                                        FB_Bacnet.StartStopCommand_145.bEnWrite := TRUE;
                                        FB_Bacnet.StartStopCommand_145.bVal := TRUE;
                                    19: 
                                        
                                        FB_Bacnet.StartStopCommand_146.bEnWrite := TRUE;
                                        FB_Bacnet.StartStopCommand_146.bVal := TRUE;
                                    20: 
                                        
                                        FB_Bacnet.StartStopCommand_147.bEnWrite := TRUE;
                                        FB_Bacnet.StartStopCommand_147.bVal := TRUE;
                                    21: 
                                        
                                        FB_Bacnet.StartStopCommand_148.bEnWrite := TRUE;
                                        FB_Bacnet.StartStopCommand_148.bVal := TRUE;
                                    22: 
                                        
                                        FB_Bacnet.StartStopCommand_176.bEnWrite := TRUE;
                                        FB_Bacnet.StartStopCommand_176.bVal := TRUE;
                                    23: 
                                        //FB_Bacnet.StartStopCommand_177.bEnWrite := TRUE;
                                        //FB_Bacnet.StartStopCommand_177.bVal := TRUE;
                                END_CASE
                            END_IF
                        END_FOR
                    END_IF
                    // Schedule Unit OFF
                    IF wSchedWEHourEndF2_ = currH AND wSchedWEMinEndF2_ = currM AND NOT bUnitTriggered THEN
                        bUnitTriggered := TRUE;
                        FOR i := 1 TO 23 DO
                            // Send command unit OFF
                            IF bUnitF2_[i] THEN 
                                CASE i OF
                                    1: 
                                        
                                        FB_Bacnet.StartStopCommand_128.bEnWrite := TRUE;
                                        FB_Bacnet.StartStopCommand_128.bVal := FALSE;
                                    2: 
                                        
                                        FB_Bacnet.StartStopCommand_129.bEnWrite := TRUE;
                                        FB_Bacnet.StartStopCommand_129.bVal := FALSE;
                                    3: 
                                        
                                        FB_Bacnet.StartStopCommand_130.bEnWrite := TRUE;
                                        FB_Bacnet.StartStopCommand_130.bVal := FALSE;
                                    4: 
                                        
                                        FB_Bacnet.StartStopCommand_131.bEnWrite := TRUE;
                                        FB_Bacnet.StartStopCommand_131.bVal := FALSE;
                                    5: 
                                        
                                        FB_Bacnet.StartStopCommand_132.bEnWrite := TRUE;
                                        FB_Bacnet.StartStopCommand_132.bVal := FALSE;
                                    6: 
                                        
                                        FB_Bacnet.StartStopCommand_133.bEnWrite := TRUE;
                                        FB_Bacnet.StartStopCommand_133.bVal := FALSE;
                                    7: 
                                        
                                        FB_Bacnet.StartStopCommand_134.bEnWrite := TRUE;
                                        FB_Bacnet.StartStopCommand_134.bVal := FALSE;
                                    8: 
                                        
                                        FB_Bacnet.StartStopCommand_135.bEnWrite := TRUE;
                                        FB_Bacnet.StartStopCommand_135.bVal := FALSE;
                                    9: 
                                        
                                        FB_Bacnet.StartStopCommand_136.bEnWrite := TRUE;
                                        FB_Bacnet.StartStopCommand_136.bVal := FALSE;
                                    10: 
                                        
                                        FB_Bacnet.StartStopCommand_137.bEnWrite := TRUE;
                                        FB_Bacnet.StartStopCommand_137.bVal := FALSE;
                                    11: 
                                        
                                        FB_Bacnet.StartStopCommand_138.bEnWrite := TRUE;
                                        FB_Bacnet.StartStopCommand_138.bVal := FALSE;
                                    12: 
                                        
                                        FB_Bacnet.StartStopCommand_139.bEnWrite := TRUE;
                                        FB_Bacnet.StartStopCommand_139.bVal := FALSE;
                                    13: 
                                        //FB_Bacnet.StartStopCommand_140.bEnWrite := TRUE;
                                        //FB_Bacnet.StartStopCommand_140.bVal := FALSE;
                                    14: 
                                        
                                        FB_Bacnet.StartStopCommand_141.bEnWrite := TRUE;
                                        FB_Bacnet.StartStopCommand_141.bVal := FALSE;
                                    15: 
                                        
                                        FB_Bacnet.StartStopCommand_142.bEnWrite := TRUE;
                                        FB_Bacnet.StartStopCommand_142.bVal := FALSE;
                                    16: 
                                        
                                        FB_Bacnet.StartStopCommand_143.bEnWrite := TRUE;
                                        FB_Bacnet.StartStopCommand_143.bVal := FALSE;
                                    17: 
                                        
                                        FB_Bacnet.StartStopCommand_144.bEnWrite := TRUE;
                                        FB_Bacnet.StartStopCommand_144.bVal := FALSE;
                                    18: 
                                        
                                        FB_Bacnet.StartStopCommand_145.bEnWrite := TRUE;
                                        FB_Bacnet.StartStopCommand_145.bVal := FALSE;
                                    19: 
                                        
                                        FB_Bacnet.StartStopCommand_146.bEnWrite := TRUE;
                                        FB_Bacnet.StartStopCommand_146.bVal := FALSE;
                                    20: 
                                        
                                        FB_Bacnet.StartStopCommand_147.bEnWrite := TRUE;
                                        FB_Bacnet.StartStopCommand_147.bVal := FALSE;
                                    21: 
                                        
                                        FB_Bacnet.StartStopCommand_148.bEnWrite := TRUE;
                                        FB_Bacnet.StartStopCommand_148.bVal := FALSE;
                                    22: 
                                        
                                        FB_Bacnet.StartStopCommand_176.bEnWrite := TRUE;
                                        FB_Bacnet.StartStopCommand_176.bVal := FALSE;
                                    23: 
                                        //FB_Bacnet.StartStopCommand_177.bEnWrite := TRUE;
                                        //FB_Bacnet.StartStopCommand_177.bVal := FALSE;
                                END_CASE
                            END_IF
                        END_FOR
                    END_IF
                END_IF
            END_IF
        END_IF

END_FUNCTION_BLOCK

// ---- POUs/FB_Scheduler/FB_Scheduler_F3.TcPOU

      FUNCTION_BLOCK FB_Scheduler_F3
      VAR_INPUT
          currH : WORD;
          currM : WORD;
          currD : WORD;
      END_VAR
      VAR_IN_OUT
          FB_Bacnet : FB_BACnet_DAIKIN_MasterStation_III_No_1;
      END_VAR
      VAR
          i : INT;
          bUnitTriggered : BOOL := FALSE; // New flag to track execution
          prevMinute : WORD := 0;        // New variable to track the previous minute
      END_VAR
      VAR PERSISTENT
          //scheduler var
          bEnSchedF3_ : BOOL := FALSE;
          wSchedWDHourStartF3_ : WORD; 
          wSchedWDMinStartF3_ : WORD; 
          wSchedWEHourStartF3_ : WORD; 
          wSchedWEMinStartF3_ : WORD;
          wSchedWDHourEndF3_ : WORD;
          wSchedWDMinEndF3_ : WORD;
          wSchedWEHourEndF3_ : WORD;
          wSchedWEMinEndF3_ : WORD;
          //unit var
          bUnitF3_ : ARRAY [1..22] OF BOOL;
      END_VAR


        // Reset trigger flag at minute change or at the exact scheduled time
        IF currM <> prevMinute OR 
           (currH = wSchedWDHourStartF3_ AND currM = wSchedWDMinStartF3_) OR 
           (currH = wSchedWDHourEndF3_ AND currM = wSchedWDMinEndF3_) THEN
            bUnitTriggered := FALSE;
            prevMinute := currM;
        END_IF

        // Unit Schedule Enable
        IF bEnSchedF3_ THEN
            // Weekday schedule
            IF currD >= 1 AND currD <= 5 THEN
                IF (wSchedWDHourStartF3_ <> wSchedWDHourEndF3_ OR wSchedWDMinStartF3_ <> wSchedWDMinEndF3_) THEN
                    // Schedule Unit ON
                    IF wSchedWDHourStartF3_ = currH AND wSchedWDMinStartF3_ = currM AND NOT bUnitTriggered THEN
                        bUnitTriggered := TRUE;
                        FOR i := 1 TO 22 DO
                            // Send command unit ON
                            IF bUnitF3_[i] THEN 
                                CASE i OF
                                    1: 

                                        //FB_Bacnet.StartStopCommand_192.bEnWrite := TRUE;
                                        //FB_Bacnet.StartStopCommand_192.bVal := TRUE;
                                    2: 
                                        
                                        FB_Bacnet.StartStopCommand_193.bEnWrite := TRUE;
                                        FB_Bacnet.StartStopCommand_193.bVal := TRUE;
                                    3: 
                                        
                                        FB_Bacnet.StartStopCommand_194.bEnWrite := TRUE;
                                        FB_Bacnet.StartStopCommand_194.bVal := TRUE;
                                    4: 
                                        
                                        FB_Bacnet.StartStopCommand_195.bEnWrite := TRUE;
                                        FB_Bacnet.StartStopCommand_195.bVal := TRUE;
                                    5: 
                                        
                                        FB_Bacnet.StartStopCommand_196.bEnWrite := TRUE;
                                        FB_Bacnet.StartStopCommand_196.bVal := TRUE;
                                    6: 
                                        
                                        FB_Bacnet.StartStopCommand_197.bEnWrite := TRUE;
                                        FB_Bacnet.StartStopCommand_197.bVal := TRUE;
                                    7: 
                                        
                                        FB_Bacnet.StartStopCommand_198.bEnWrite := TRUE;
                                        FB_Bacnet.StartStopCommand_198.bVal := TRUE;
                                    8: 
                                        
                                        FB_Bacnet.StartStopCommand_199.bEnWrite := TRUE;
                                        FB_Bacnet.StartStopCommand_199.bVal := TRUE;
                                    9: 
                                        
                                        FB_Bacnet.StartStopCommand_200.bEnWrite := TRUE;
                                        FB_Bacnet.StartStopCommand_200.bVal := TRUE;
                                    10: 
                                        
                                        FB_Bacnet.StartStopCommand_201.bEnWrite := TRUE;
                                        FB_Bacnet.StartStopCommand_201.bVal := TRUE;
                                    11: 
                                        
                                        FB_Bacnet.StartStopCommand_202.bEnWrite := TRUE;
                                        FB_Bacnet.StartStopCommand_202.bVal := TRUE;
                                    12: 
                                        
                                        FB_Bacnet.StartStopCommand_203.bEnWrite := TRUE;
                                        FB_Bacnet.StartStopCommand_203.bVal := TRUE;
                                    13: 
                                        
                                        FB_Bacnet.StartStopCommand_204.bEnWrite := TRUE;
                                        FB_Bacnet.StartStopCommand_204.bVal := TRUE;
                                    14: 
                                        
                                        FB_Bacnet.StartStopCommand_205.bEnWrite := TRUE;
                                        FB_Bacnet.StartStopCommand_205.bVal := TRUE;
                                    15: 
                                        
                                        FB_Bacnet.StartStopCommand_206.bEnWrite := TRUE;
                                        FB_Bacnet.StartStopCommand_206.bVal := TRUE;
                                    16: 
                                        
                                        FB_Bacnet.StartStopCommand_207.bEnWrite := TRUE;
                                        FB_Bacnet.StartStopCommand_207.bVal := TRUE;
                                    17: 
                                        
                                        FB_Bacnet.StartStopCommand_208.bEnWrite := TRUE;
                                        FB_Bacnet.StartStopCommand_208.bVal := TRUE;
                                    18: 
                                        
                                        FB_Bacnet.StartStopCommand_209.bEnWrite := TRUE;
                                        FB_Bacnet.StartStopCommand_209.bVal := TRUE;
                                    19: 
                                        
                                        FB_Bacnet.StartStopCommand_210.bEnWrite := TRUE;
                                        FB_Bacnet.StartStopCommand_210.bVal := TRUE;
                                    20: 
                                        
                                        FB_Bacnet.StartStopCommand_211.bEnWrite := TRUE;
                                        FB_Bacnet.StartStopCommand_211.bVal := TRUE;
                                    21: 
                                        
                                        FB_Bacnet.StartStopCommand_212.bEnWrite := TRUE;
                                        FB_Bacnet.StartStopCommand_212.bVal := TRUE;
                                    22: 
                                        
                                        FB_Bacnet.StartStopCommand_224.bEnWrite := TRUE;
                                        FB_Bacnet.StartStopCommand_224.bVal := TRUE;
                                END_CASE
                            END_IF
                        END_FOR
                    END_IF
                    // Schedule Unit OFF
                    IF wSchedWDHourEndF3_ = currH AND wSchedWDMinEndF3_ = currM AND NOT bUnitTriggered THEN
                        bUnitTriggered := TRUE;
                        FOR i := 1 TO 22 DO
                            // Send command unit OFF
                            IF bUnitF3_[i] THEN 
                                CASE i OF
                                    1: 

                                        //FB_Bacnet.StartStopCommand_192.bEnWrite := TRUE;
                                        //FB_Bacnet.StartStopCommand_192.bVal := FALSE;
                                    2: 
                                        
                                        FB_Bacnet.StartStopCommand_193.bEnWrite := TRUE;
                                        FB_Bacnet.StartStopCommand_193.bVal := FALSE;
                                    3: 
                                        
                                        FB_Bacnet.StartStopCommand_194.bEnWrite := TRUE;
                                        FB_Bacnet.StartStopCommand_194.bVal := FALSE;
                                    4: 
                                        
                                        FB_Bacnet.StartStopCommand_195.bEnWrite := TRUE;
                                        FB_Bacnet.StartStopCommand_195.bVal := FALSE;
                                    5: 
                                        
                                        FB_Bacnet.StartStopCommand_196.bEnWrite := TRUE;
                                        FB_Bacnet.StartStopCommand_196.bVal := FALSE;
                                    6: 
                                        
                                        FB_Bacnet.StartStopCommand_197.bEnWrite := TRUE;
                                        FB_Bacnet.StartStopCommand_197.bVal := FALSE;
                                    7: 
                                        
                                        FB_Bacnet.StartStopCommand_198.bEnWrite := TRUE;
                                        FB_Bacnet.StartStopCommand_198.bVal := FALSE;
                                    8: 
                                        
                                        FB_Bacnet.StartStopCommand_199.bEnWrite := TRUE;
                                        FB_Bacnet.StartStopCommand_199.bVal := FALSE;
                                    9: 
                                        
                                        FB_Bacnet.StartStopCommand_200.bEnWrite := TRUE;
                                        FB_Bacnet.StartStopCommand_200.bVal := FALSE;
                                    10: 
                                        
                                        FB_Bacnet.StartStopCommand_201.bEnWrite := TRUE;
                                        FB_Bacnet.StartStopCommand_201.bVal := FALSE;
                                    11: 
                                        
                                        FB_Bacnet.StartStopCommand_202.bEnWrite := TRUE;
                                        FB_Bacnet.StartStopCommand_202.bVal := FALSE;
                                    12: 
                                        
                                        FB_Bacnet.StartStopCommand_203.bEnWrite := TRUE;
                                        FB_Bacnet.StartStopCommand_203.bVal := FALSE;
                                    13: 
                                        
                                        FB_Bacnet.StartStopCommand_204.bEnWrite := TRUE;
                                        FB_Bacnet.StartStopCommand_204.bVal := FALSE;
                                    14: 
                                        
                                        FB_Bacnet.StartStopCommand_205.bEnWrite := TRUE;
                                        FB_Bacnet.StartStopCommand_205.bVal := FALSE;
                                    15: 
                                        
                                        FB_Bacnet.StartStopCommand_206.bEnWrite := TRUE;
                                        FB_Bacnet.StartStopCommand_206.bVal := FALSE;
                                    16: 
                                        
                                        FB_Bacnet.StartStopCommand_207.bEnWrite := TRUE;
                                        FB_Bacnet.StartStopCommand_207.bVal := FALSE;
                                    17: 
                                        
                                        FB_Bacnet.StartStopCommand_208.bEnWrite := TRUE;
                                        FB_Bacnet.StartStopCommand_208.bVal := FALSE;
                                    18: 
                                        
                                        FB_Bacnet.StartStopCommand_209.bEnWrite := TRUE;
                                        FB_Bacnet.StartStopCommand_209.bVal := FALSE;
                                    19: 
                                        
                                        FB_Bacnet.StartStopCommand_210.bEnWrite := TRUE;
                                        FB_Bacnet.StartStopCommand_210.bVal := FALSE;
                                    20: 
                                        
                                        FB_Bacnet.StartStopCommand_211.bEnWrite := TRUE;
                                        FB_Bacnet.StartStopCommand_211.bVal := FALSE;
                                    21: 
                                        
                                        FB_Bacnet.StartStopCommand_212.bEnWrite := TRUE;
                                        FB_Bacnet.StartStopCommand_212.bVal := FALSE;
                                    22: 
                                        
                                        FB_Bacnet.StartStopCommand_224.bEnWrite := TRUE;
                                        FB_Bacnet.StartStopCommand_224.bVal := FALSE;
                                END_CASE
                            END_IF
                        END_FOR
                    END_IF
                END_IF
            END_IF

            // Weekend schedule
            IF currD = 0 OR currD = 6 THEN
                IF (wSchedWEHourStartF3_ <> wSchedWEHourEndF3_ OR wSchedWEMinStartF3_ <> wSchedWEMinEndF3_) THEN
                    // Schedule Unit ON
                    IF wSchedWEHourStartF3_ = currH AND wSchedWEMinStartF3_ = currM AND NOT bUnitTriggered THEN
                        bUnitTriggered := TRUE;
                        FOR i := 1 TO 22 DO
                            // Send command unit ON
                            IF bUnitF3_[i] THEN 
                                CASE i OF
                                    1: 

                                        //FB_Bacnet.StartStopCommand_192.bEnWrite := TRUE;
                                        //FB_Bacnet.StartStopCommand_192.bVal := TRUE;
                                    2: 
                                        
                                        FB_Bacnet.StartStopCommand_193.bEnWrite := TRUE;
                                        FB_Bacnet.StartStopCommand_193.bVal := TRUE;
                                    3: 
                                        
                                        FB_Bacnet.StartStopCommand_194.bEnWrite := TRUE;
                                        FB_Bacnet.StartStopCommand_194.bVal := TRUE;
                                    4: 
                                        
                                        FB_Bacnet.StartStopCommand_195.bEnWrite := TRUE;
                                        FB_Bacnet.StartStopCommand_195.bVal := TRUE;
                                    5: 
                                        
                                        FB_Bacnet.StartStopCommand_196.bEnWrite := TRUE;
                                        FB_Bacnet.StartStopCommand_196.bVal := TRUE;
                                    6: 
                                        
                                        FB_Bacnet.StartStopCommand_197.bEnWrite := TRUE;
                                        FB_Bacnet.StartStopCommand_197.bVal := TRUE;
                                    7: 
                                        
                                        FB_Bacnet.StartStopCommand_198.bEnWrite := TRUE;
                                        FB_Bacnet.StartStopCommand_198.bVal := TRUE;
                                    8: 
                                        
                                        FB_Bacnet.StartStopCommand_199.bEnWrite := TRUE;
                                        FB_Bacnet.StartStopCommand_199.bVal := TRUE;
                                    9: 
                                        
                                        FB_Bacnet.StartStopCommand_200.bEnWrite := TRUE;
                                        FB_Bacnet.StartStopCommand_200.bVal := TRUE;
                                    10: 
                                        
                                        FB_Bacnet.StartStopCommand_201.bEnWrite := TRUE;
                                        FB_Bacnet.StartStopCommand_201.bVal := TRUE;
                                    11: 
                                        
                                        FB_Bacnet.StartStopCommand_202.bEnWrite := TRUE;
                                        FB_Bacnet.StartStopCommand_202.bVal := TRUE;
                                    12: 
                                        
                                        FB_Bacnet.StartStopCommand_203.bEnWrite := TRUE;
                                        FB_Bacnet.StartStopCommand_203.bVal := TRUE;
                                    13: 
                                        
                                        FB_Bacnet.StartStopCommand_204.bEnWrite := TRUE;
                                        FB_Bacnet.StartStopCommand_204.bVal := TRUE;
                                    14: 
                                        
                                        FB_Bacnet.StartStopCommand_205.bEnWrite := TRUE;
                                        FB_Bacnet.StartStopCommand_205.bVal := TRUE;
                                    15: 
                                        
                                        FB_Bacnet.StartStopCommand_206.bEnWrite := TRUE;
                                        FB_Bacnet.StartStopCommand_206.bVal := TRUE;
                                    16: 
                                        
                                        FB_Bacnet.StartStopCommand_207.bEnWrite := TRUE;
                                        FB_Bacnet.StartStopCommand_207.bVal := TRUE;
                                    17: 
                                        
                                        FB_Bacnet.StartStopCommand_208.bEnWrite := TRUE;
                                        FB_Bacnet.StartStopCommand_208.bVal := TRUE;
                                    18: 
                                        
                                        FB_Bacnet.StartStopCommand_209.bEnWrite := TRUE;
                                        FB_Bacnet.StartStopCommand_209.bVal := TRUE;
                                    19: 
                                        
                                        FB_Bacnet.StartStopCommand_210.bEnWrite := TRUE;
                                        FB_Bacnet.StartStopCommand_210.bVal := TRUE;
                                    20: 
                                        
                                        FB_Bacnet.StartStopCommand_211.bEnWrite := TRUE;
                                        FB_Bacnet.StartStopCommand_211.bVal := TRUE;
                                    21: 
                                        
                                        FB_Bacnet.StartStopCommand_212.bEnWrite := TRUE;
                                        FB_Bacnet.StartStopCommand_212.bVal := TRUE;
                                    22: 
                                        
                                        FB_Bacnet.StartStopCommand_224.bEnWrite := TRUE;
                                        FB_Bacnet.StartStopCommand_224.bVal := TRUE;
                                END_CASE
                            END_IF
                        END_FOR
                    END_IF
                    // Schedule Unit OFF
                    IF wSchedWEHourEndF3_ = currH AND wSchedWEMinEndF3_ = currM AND NOT bUnitTriggered THEN
                        bUnitTriggered := TRUE;
                        FOR i := 1 TO 22 DO
                            // Send command unit OFF
                            IF bUnitF3_[i] THEN 
                                CASE i OF
                                    1: 

                                        //FB_Bacnet.StartStopCommand_192.bEnWrite := TRUE;
                                        //FB_Bacnet.StartStopCommand_192.bVal := FALSE;
                                    2: 
                                        
                                        FB_Bacnet.StartStopCommand_193.bEnWrite := TRUE;
                                        FB_Bacnet.StartStopCommand_193.bVal := FALSE;
                                    3: 
                                        
                                        FB_Bacnet.StartStopCommand_194.bEnWrite := TRUE;
                                        FB_Bacnet.StartStopCommand_194.bVal := FALSE;
                                    4: 
                                        
                                        FB_Bacnet.StartStopCommand_195.bEnWrite := TRUE;
                                        FB_Bacnet.StartStopCommand_195.bVal := FALSE;
                                    5: 
                                        
                                        FB_Bacnet.StartStopCommand_196.bEnWrite := TRUE;
                                        FB_Bacnet.StartStopCommand_196.bVal := FALSE;
                                    6: 
                                        
                                        FB_Bacnet.StartStopCommand_197.bEnWrite := TRUE;
                                        FB_Bacnet.StartStopCommand_197.bVal := FALSE;
                                    7: 
                                        
                                        FB_Bacnet.StartStopCommand_198.bEnWrite := TRUE;
                                        FB_Bacnet.StartStopCommand_198.bVal := FALSE;
                                    8: 
                                        
                                        FB_Bacnet.StartStopCommand_199.bEnWrite := TRUE;
                                        FB_Bacnet.StartStopCommand_199.bVal := FALSE;
                                    9: 
                                        
                                        FB_Bacnet.StartStopCommand_200.bEnWrite := TRUE;
                                        FB_Bacnet.StartStopCommand_200.bVal := FALSE;
                                    10: 
                                        
                                        FB_Bacnet.StartStopCommand_201.bEnWrite := TRUE;
                                        FB_Bacnet.StartStopCommand_201.bVal := FALSE;
                                    11: 
                                        
                                        FB_Bacnet.StartStopCommand_202.bEnWrite := TRUE;
                                        FB_Bacnet.StartStopCommand_202.bVal := FALSE;
                                    12: 
                                        
                                        FB_Bacnet.StartStopCommand_203.bEnWrite := TRUE;
                                        FB_Bacnet.StartStopCommand_203.bVal := FALSE;
                                    13: 
                                        
                                        FB_Bacnet.StartStopCommand_204.bEnWrite := TRUE;
                                        FB_Bacnet.StartStopCommand_204.bVal := FALSE;
                                    14: 
                                        
                                        FB_Bacnet.StartStopCommand_205.bEnWrite := TRUE;
                                        FB_Bacnet.StartStopCommand_205.bVal := FALSE;
                                    15: 
                                        
                                        FB_Bacnet.StartStopCommand_206.bEnWrite := TRUE;
                                        FB_Bacnet.StartStopCommand_206.bVal := FALSE;
                                    16: 
                                        
                                        FB_Bacnet.StartStopCommand_207.bEnWrite := TRUE;
                                        FB_Bacnet.StartStopCommand_207.bVal := FALSE;
                                    17: 
                                        
                                        FB_Bacnet.StartStopCommand_208.bEnWrite := TRUE;
                                        FB_Bacnet.StartStopCommand_208.bVal := FALSE;
                                    18: 
                                        
                                        FB_Bacnet.StartStopCommand_209.bEnWrite := TRUE;
                                        FB_Bacnet.StartStopCommand_209.bVal := FALSE;
                                    19: 
                                        
                                        FB_Bacnet.StartStopCommand_210.bEnWrite := TRUE;
                                        FB_Bacnet.StartStopCommand_210.bVal := FALSE;
                                    20: 
                                        
                                        FB_Bacnet.StartStopCommand_211.bEnWrite := TRUE;
                                        FB_Bacnet.StartStopCommand_211.bVal := FALSE;
                                    21: 
                                        
                                        FB_Bacnet.StartStopCommand_212.bEnWrite := TRUE;
                                        FB_Bacnet.StartStopCommand_212.bVal := FALSE;
                                    22: 
                                        
                                        FB_Bacnet.StartStopCommand_224.bEnWrite := TRUE;
                                        FB_Bacnet.StartStopCommand_224.bVal := FALSE;
                                END_CASE
                            END_IF
                        END_FOR
                    END_IF
                END_IF
            END_IF
        END_IF

END_FUNCTION_BLOCK

// ---- POUs/FB_Scheduler/FB_Scheduler_F5.TcPOU

      FUNCTION_BLOCK FB_Scheduler_F5
      VAR_INPUT
          currH : WORD;
          currM : WORD;
          currD : WORD;
      END_VAR
      VAR_IN_OUT
          FB_Bacnet : FB_BACnet_DAIKIN_MasterStation_III_No_2;
          FB_Bacnet_b : FB_BACnet_DAIKIN_MasterStation_III_No_1;
      END_VAR
      VAR
          i : INT;
          bUnitTriggered : BOOL := FALSE; // New flag to track execution
          prevMinute : WORD := 0;        // New variable to track the previous minute
      END_VAR
      VAR PERSISTENT
          //scheduler var
          bEnSchedF5_ : BOOL := FALSE;
          wSchedWDHourStartF5_ : WORD; 
          wSchedWDMinStartF5_ : WORD; 
          wSchedWEHourStartF5_ : WORD; 
          wSchedWEMinStartF5_ : WORD;
          wSchedWDHourEndF5_ : WORD;
          wSchedWDMinEndF5_ : WORD;
          wSchedWEHourEndF5_ : WORD;
          wSchedWEMinEndF5_ : WORD;
          //unit var
          bUnitF5_ : ARRAY [1..22] OF BOOL;
      END_VAR


        // Reset trigger flag at minute change or at the exact scheduled time
        IF currM <> prevMinute OR 
           (currH = wSchedWDHourStartF5_ AND currM = wSchedWDMinStartF5_) OR 
           (currH = wSchedWDHourEndF5_ AND currM = wSchedWDMinEndF5_) THEN
            bUnitTriggered := FALSE;
            prevMinute := currM;
        END_IF

        // Unit Schedule Enable
        IF bEnSchedF5_ THEN
            // Weekday schedule
            IF currD >= 1 AND currD <= 5 THEN
                IF (wSchedWDHourStartF5_ <> wSchedWDHourEndF5_ OR wSchedWDMinStartF5_ <> wSchedWDMinEndF5_) THEN
                    // Schedule Unit ON
                    IF wSchedWDHourStartF5_ = currH AND wSchedWDMinStartF5_ = currM AND NOT bUnitTriggered THEN
                        bUnitTriggered := TRUE;
                        FOR i := 1 TO 22 DO
                            // Send command unit ON
                            IF bUnitF5_[i] THEN 
                                CASE i OF
                                    1: 
                                        
                                        FB_Bacnet.StartStopCommand_000.bEnWrite := TRUE;
                                        FB_Bacnet.StartStopCommand_000.bVal := TRUE;
                                    2: 
                                        
                                        FB_Bacnet.StartStopCommand_001.bEnWrite := TRUE;
                                        FB_Bacnet.StartStopCommand_001.bVal := TRUE;
                                    3: 
                                        
                                        FB_Bacnet.StartStopCommand_002.bEnWrite := TRUE;
                                        FB_Bacnet.StartStopCommand_002.bVal := TRUE;
                                    4: 
                                        
                                        FB_Bacnet.StartStopCommand_003.bEnWrite := TRUE;
                                        FB_Bacnet.StartStopCommand_003.bVal := TRUE;
                                    5: 
                                        
                                        FB_Bacnet.StartStopCommand_004.bEnWrite := TRUE;
                                        FB_Bacnet.StartStopCommand_004.bVal := TRUE;
                                    6: 
                                        
                                        FB_Bacnet.StartStopCommand_005.bEnWrite := TRUE;
                                        FB_Bacnet.StartStopCommand_005.bVal := TRUE;
                                    7: 
                                        
                                        FB_Bacnet.StartStopCommand_006.bEnWrite := TRUE;
                                        FB_Bacnet.StartStopCommand_006.bVal := TRUE;
                                    8: 
                                        
                                        FB_Bacnet.StartStopCommand_007.bEnWrite := TRUE;
                                        FB_Bacnet.StartStopCommand_007.bVal := TRUE;
                                    9: 
                                        
                                        FB_Bacnet.StartStopCommand_008.bEnWrite := TRUE;
                                        FB_Bacnet.StartStopCommand_008.bVal := TRUE;
                                    10: 
                                        
                                        FB_Bacnet.StartStopCommand_009.bEnWrite := TRUE;
                                        FB_Bacnet.StartStopCommand_009.bVal := TRUE;
                                    11: 
                                        
                                        FB_Bacnet.StartStopCommand_010.bEnWrite := TRUE;
                                        FB_Bacnet.StartStopCommand_010.bVal := TRUE;
                                    12: 
                                        
                                        FB_Bacnet.StartStopCommand_011.bEnWrite := TRUE;
                                        FB_Bacnet.StartStopCommand_011.bVal := TRUE;
                                    13: 
                                        
                                        FB_Bacnet.StartStopCommand_012.bEnWrite := TRUE;
                                        FB_Bacnet.StartStopCommand_012.bVal := TRUE;
                                    14: 
                                        
                                        FB_Bacnet.StartStopCommand_013.bEnWrite := TRUE;
                                        FB_Bacnet.StartStopCommand_013.bVal := TRUE;
                                    15: 
                                        
                                        FB_Bacnet.StartStopCommand_014.bEnWrite := TRUE;
                                        FB_Bacnet.StartStopCommand_014.bVal := TRUE;
                                    16: 
                                        
                                        FB_Bacnet.StartStopCommand_015.bEnWrite := TRUE;
                                        FB_Bacnet.StartStopCommand_015.bVal := TRUE;
                                    17: 
                                        
                                        FB_Bacnet.StartStopCommand_016.bEnWrite := TRUE;
                                        FB_Bacnet.StartStopCommand_016.bVal := TRUE;
                                    18: 
                                        
                                        FB_Bacnet.StartStopCommand_017.bEnWrite := TRUE;
                                        FB_Bacnet.StartStopCommand_017.bVal := TRUE;
                                    19: 
                                        
                                        FB_Bacnet.StartStopCommand_018.bEnWrite := TRUE;
                                        FB_Bacnet.StartStopCommand_018.bVal := TRUE;
                                    20: 
                                        
                                        FB_Bacnet.StartStopCommand_019.bEnWrite := TRUE;
                                        FB_Bacnet.StartStopCommand_019.bVal := TRUE;
                                    21: 
                                        
                                        FB_Bacnet.StartStopCommand_020.bEnWrite := TRUE;
                                        FB_Bacnet.StartStopCommand_020.bVal := TRUE;
                                    22: 
                                        
                                        FB_Bacnet_b.StartStopCommand_225.bEnWrite := TRUE;
                                        FB_Bacnet_b.StartStopCommand_225.bVal := TRUE;
                                END_CASE
                            END_IF
                        END_FOR
                    END_IF
                    // Schedule Unit OFF
                    IF wSchedWDHourEndF5_ = currH AND wSchedWDMinEndF5_ = currM AND NOT bUnitTriggered THEN
                        bUnitTriggered := TRUE;
                        FOR i := 1 TO 22 DO
                            // Send command unit OFF
                            IF bUnitF5_[i] THEN 
                                CASE i OF
                                    1: 
                                        
                                        FB_Bacnet.StartStopCommand_000.bEnWrite := TRUE;
                                        FB_Bacnet.StartStopCommand_000.bVal := FALSE;
                                    2: 
                                        
                                        FB_Bacnet.StartStopCommand_001.bEnWrite := TRUE;
                                        FB_Bacnet.StartStopCommand_001.bVal := FALSE;
                                    3: 
                                        
                                        FB_Bacnet.StartStopCommand_002.bEnWrite := TRUE;
                                        FB_Bacnet.StartStopCommand_002.bVal := FALSE;
                                    4: 
                                        
                                        FB_Bacnet.StartStopCommand_003.bEnWrite := TRUE;
                                        FB_Bacnet.StartStopCommand_003.bVal := FALSE;
                                    5: 
                                        
                                        FB_Bacnet.StartStopCommand_004.bEnWrite := TRUE;
                                        FB_Bacnet.StartStopCommand_004.bVal := FALSE;
                                    6: 
                                        
                                        FB_Bacnet.StartStopCommand_005.bEnWrite := TRUE;
                                        FB_Bacnet.StartStopCommand_005.bVal := FALSE;
                                    7: 
                                        
                                        FB_Bacnet.StartStopCommand_006.bEnWrite := TRUE;
                                        FB_Bacnet.StartStopCommand_006.bVal := FALSE;
                                    8: 
                                        
                                        FB_Bacnet.StartStopCommand_007.bEnWrite := TRUE;
                                        FB_Bacnet.StartStopCommand_007.bVal := FALSE;
                                    9: 
                                        
                                        FB_Bacnet.StartStopCommand_008.bEnWrite := TRUE;
                                        FB_Bacnet.StartStopCommand_008.bVal := FALSE;
                                    10: 
                                        
                                        FB_Bacnet.StartStopCommand_009.bEnWrite := TRUE;
                                        FB_Bacnet.StartStopCommand_009.bVal := FALSE;
                                    11: 
                                        
                                        FB_Bacnet.StartStopCommand_010.bEnWrite := TRUE;
                                        FB_Bacnet.StartStopCommand_010.bVal := FALSE;
                                    12: 
                                        
                                        FB_Bacnet.StartStopCommand_011.bEnWrite := TRUE;
                                        FB_Bacnet.StartStopCommand_011.bVal := FALSE;
                                    13: 
                                        
                                        FB_Bacnet.StartStopCommand_012.bEnWrite := TRUE;
                                        FB_Bacnet.StartStopCommand_012.bVal := FALSE;
                                    14: 
                                        
                                        FB_Bacnet.StartStopCommand_013.bEnWrite := TRUE;
                                        FB_Bacnet.StartStopCommand_013.bVal := FALSE;
                                    15: 
                                        
                                        FB_Bacnet.StartStopCommand_014.bEnWrite := TRUE;
                                        FB_Bacnet.StartStopCommand_014.bVal := FALSE;
                                    16: 
                                        
                                        FB_Bacnet.StartStopCommand_015.bEnWrite := TRUE;
                                        FB_Bacnet.StartStopCommand_015.bVal := FALSE;
                                    17: 
                                        
                                        FB_Bacnet.StartStopCommand_016.bEnWrite := TRUE;
                                        FB_Bacnet.StartStopCommand_016.bVal := FALSE;
                                    18: 
                                        
                                        FB_Bacnet.StartStopCommand_017.bEnWrite := TRUE;
                                        FB_Bacnet.StartStopCommand_017.bVal := FALSE;
                                    19: 
                                        
                                        FB_Bacnet.StartStopCommand_018.bEnWrite := TRUE;
                                        FB_Bacnet.StartStopCommand_018.bVal := FALSE;
                                    20: 
                                        
                                        FB_Bacnet.StartStopCommand_019.bEnWrite := TRUE;
                                        FB_Bacnet.StartStopCommand_019.bVal := FALSE;
                                    21: 
                                        
                                        FB_Bacnet.StartStopCommand_020.bEnWrite := TRUE;
                                        FB_Bacnet.StartStopCommand_020.bVal := FALSE;
                                    22: 
                                        
                                        FB_Bacnet_b.StartStopCommand_225.bEnWrite := TRUE;
                                        FB_Bacnet_b.StartStopCommand_225.bVal := FALSE;
                                END_CASE
                            END_IF
                        END_FOR
                    END_IF
                END_IF
            END_IF

            // Weekend schedule
            IF currD = 0 OR currD = 6 THEN
                IF (wSchedWEHourStartF5_ <> wSchedWEHourEndF5_ OR wSchedWEMinStartF5_ <> wSchedWEMinEndF5_) THEN
                    // Schedule Unit ON
                    IF wSchedWEHourStartF5_ = currH AND wSchedWEMinStartF5_ = currM AND NOT bUnitTriggered THEN
                        bUnitTriggered := TRUE;
                        FOR i := 1 TO 22 DO
                            // Send command unit ON
                            IF bUnitF5_[i] THEN 
                                CASE i OF
                                    1: 
                                        
                                        FB_Bacnet.StartStopCommand_000.bEnWrite := TRUE;
                                        FB_Bacnet.StartStopCommand_000.bVal := TRUE;
                                    2: 
                                        
                                        FB_Bacnet.StartStopCommand_001.bEnWrite := TRUE;
                                        FB_Bacnet.StartStopCommand_001.bVal := TRUE;
                                    3: 
                                        
                                        FB_Bacnet.StartStopCommand_002.bEnWrite := TRUE;
                                        FB_Bacnet.StartStopCommand_002.bVal := TRUE;
                                    4: 
                                        
                                        FB_Bacnet.StartStopCommand_003.bEnWrite := TRUE;
                                        FB_Bacnet.StartStopCommand_003.bVal := TRUE;
                                    5: 
                                        
                                        FB_Bacnet.StartStopCommand_004.bEnWrite := TRUE;
                                        FB_Bacnet.StartStopCommand_004.bVal := TRUE;
                                    6: 
                                        
                                        FB_Bacnet.StartStopCommand_005.bEnWrite := TRUE;
                                        FB_Bacnet.StartStopCommand_005.bVal := TRUE;
                                    7: 
                                        
                                        FB_Bacnet.StartStopCommand_006.bEnWrite := TRUE;
                                        FB_Bacnet.StartStopCommand_006.bVal := TRUE;
                                    8: 
                                        
                                        FB_Bacnet.StartStopCommand_007.bEnWrite := TRUE;
                                        FB_Bacnet.StartStopCommand_007.bVal := TRUE;
                                    9: 
                                        
                                        FB_Bacnet.StartStopCommand_008.bEnWrite := TRUE;
                                        FB_Bacnet.StartStopCommand_008.bVal := TRUE;
                                    10: 
                                        
                                        FB_Bacnet.StartStopCommand_009.bEnWrite := TRUE;
                                        FB_Bacnet.StartStopCommand_009.bVal := TRUE;
                                    11: 
                                        
                                        FB_Bacnet.StartStopCommand_010.bEnWrite := TRUE;
                                        FB_Bacnet.StartStopCommand_010.bVal := TRUE;
                                    12: 
                                        
                                        FB_Bacnet.StartStopCommand_011.bEnWrite := TRUE;
                                        FB_Bacnet.StartStopCommand_011.bVal := TRUE;
                                    13: 
                                        
                                        FB_Bacnet.StartStopCommand_012.bEnWrite := TRUE;
                                        FB_Bacnet.StartStopCommand_012.bVal := TRUE;
                                    14: 
                                        
                                        FB_Bacnet.StartStopCommand_013.bEnWrite := TRUE;
                                        FB_Bacnet.StartStopCommand_013.bVal := TRUE;
                                    15: 
                                        
                                        FB_Bacnet.StartStopCommand_014.bEnWrite := TRUE;
                                        FB_Bacnet.StartStopCommand_014.bVal := TRUE;
                                    16: 
                                        
                                        FB_Bacnet.StartStopCommand_015.bEnWrite := TRUE;
                                        FB_Bacnet.StartStopCommand_015.bVal := TRUE;
                                    17: 
                                        
                                        FB_Bacnet.StartStopCommand_016.bEnWrite := TRUE;
                                        FB_Bacnet.StartStopCommand_016.bVal := TRUE;
                                    18: 
                                        
                                        FB_Bacnet.StartStopCommand_017.bEnWrite := TRUE;
                                        FB_Bacnet.StartStopCommand_017.bVal := TRUE;
                                    19: 
                                        
                                        FB_Bacnet.StartStopCommand_018.bEnWrite := TRUE;
                                        FB_Bacnet.StartStopCommand_018.bVal := TRUE;
                                    20: 
                                        
                                        FB_Bacnet.StartStopCommand_019.bEnWrite := TRUE;
                                        FB_Bacnet.StartStopCommand_019.bVal := TRUE;
                                    21: 
                                        
                                        FB_Bacnet.StartStopCommand_020.bEnWrite := TRUE;
                                        FB_Bacnet.StartStopCommand_020.bVal := TRUE;
                                    22: 
                                        
                                        FB_Bacnet_b.StartStopCommand_225.bEnWrite := TRUE;
                                        FB_Bacnet_b.StartStopCommand_225.bVal := TRUE;
                                END_CASE
                            END_IF
                        END_FOR
                    END_IF
                    // Schedule Unit OFF
                    IF wSchedWEHourEndF5_ = currH AND wSchedWEMinEndF5_ = currM AND NOT bUnitTriggered THEN
                        bUnitTriggered := TRUE;
                        FOR i := 1 TO 22 DO
                            // Send command unit OFF
                            IF bUnitF5_[i] THEN 
                                CASE i OF
                                    1: 
                                        
                                        FB_Bacnet.StartStopCommand_000.bEnWrite := TRUE;
                                        FB_Bacnet.StartStopCommand_000.bVal := FALSE;
                                    2: 
                                        
                                        FB_Bacnet.StartStopCommand_001.bEnWrite := TRUE;
                                        FB_Bacnet.StartStopCommand_001.bVal := FALSE;
                                    3: 
                                        
                                        FB_Bacnet.StartStopCommand_002.bEnWrite := TRUE;
                                        FB_Bacnet.StartStopCommand_002.bVal := FALSE;
                                    4: 
                                        
                                        FB_Bacnet.StartStopCommand_003.bEnWrite := TRUE;
                                        FB_Bacnet.StartStopCommand_003.bVal := FALSE;
                                    5: 
                                        
                                        FB_Bacnet.StartStopCommand_004.bEnWrite := TRUE;
                                        FB_Bacnet.StartStopCommand_004.bVal := FALSE;
                                    6: 
                                        
                                        FB_Bacnet.StartStopCommand_005.bEnWrite := TRUE;
                                        FB_Bacnet.StartStopCommand_005.bVal := FALSE;
                                    7: 
                                        
                                        FB_Bacnet.StartStopCommand_006.bEnWrite := TRUE;
                                        FB_Bacnet.StartStopCommand_006.bVal := FALSE;
                                    8: 
                                        
                                        FB_Bacnet.StartStopCommand_007.bEnWrite := TRUE;
                                        FB_Bacnet.StartStopCommand_007.bVal := FALSE;
                                    9: 
                                        
                                        FB_Bacnet.StartStopCommand_008.bEnWrite := TRUE;
                                        FB_Bacnet.StartStopCommand_008.bVal := FALSE;
                                    10: 
                                        
                                        FB_Bacnet.StartStopCommand_009.bEnWrite := TRUE;
                                        FB_Bacnet.StartStopCommand_009.bVal := FALSE;
                                    11: 
                                        
                                        FB_Bacnet.StartStopCommand_010.bEnWrite := TRUE;
                                        FB_Bacnet.StartStopCommand_010.bVal := FALSE;
                                    12: 
                                        
                                        FB_Bacnet.StartStopCommand_011.bEnWrite := TRUE;
                                        FB_Bacnet.StartStopCommand_011.bVal := FALSE;
                                    13: 
                                        
                                        FB_Bacnet.StartStopCommand_012.bEnWrite := TRUE;
                                        FB_Bacnet.StartStopCommand_012.bVal := FALSE;
                                    14: 
                                        
                                        FB_Bacnet.StartStopCommand_013.bEnWrite := TRUE;
                                        FB_Bacnet.StartStopCommand_013.bVal := FALSE;
                                    15: 
                                        
                                        FB_Bacnet.StartStopCommand_014.bEnWrite := TRUE;
                                        FB_Bacnet.StartStopCommand_014.bVal := FALSE;
                                    16: 
                                        
                                        FB_Bacnet.StartStopCommand_015.bEnWrite := TRUE;
                                        FB_Bacnet.StartStopCommand_015.bVal := FALSE;
                                    17: 
                                        
                                        FB_Bacnet.StartStopCommand_016.bEnWrite := TRUE;
                                        FB_Bacnet.StartStopCommand_016.bVal := FALSE;
                                    18: 
                                        
                                        FB_Bacnet.StartStopCommand_017.bEnWrite := TRUE;
                                        FB_Bacnet.StartStopCommand_017.bVal := FALSE;
                                    19: 
                                        
                                        FB_Bacnet.StartStopCommand_018.bEnWrite := TRUE;
                                        FB_Bacnet.StartStopCommand_018.bVal := FALSE;
                                    20: 
                                        
                                        FB_Bacnet.StartStopCommand_019.bEnWrite := TRUE;
                                        FB_Bacnet.StartStopCommand_019.bVal := FALSE;
                                    21: 
                                        
                                        FB_Bacnet.StartStopCommand_020.bEnWrite := TRUE;
                                        FB_Bacnet.StartStopCommand_020.bVal := FALSE;
                                    22: 
                                        
                                        FB_Bacnet_b.StartStopCommand_225.bEnWrite := TRUE;
                                        FB_Bacnet_b.StartStopCommand_225.bVal := FALSE;
                                END_CASE
                            END_IF
                        END_FOR
                    END_IF
                END_IF
            END_IF
        END_IF

END_FUNCTION_BLOCK

// ---- POUs/FB_Scheduler/FB_Scheduler_F6.TcPOU

      FUNCTION_BLOCK FB_Scheduler_F6
      VAR_INPUT
          currH : WORD;
          currM : WORD;
          currD : WORD;
      END_VAR
      VAR_IN_OUT
          FB_Bacnet : FB_BACnet_DAIKIN_MasterStation_III_No_2;
          FB_Bacnet_b : FB_BACnet_DAIKIN_MasterStation_III_No_1;
      END_VAR
      VAR
          i : INT;
          bUnitTriggered : BOOL := FALSE; // New flag to track execution
          prevMinute : WORD := 0;        // New variable to track the previous minute
      END_VAR
      VAR PERSISTENT
          //scheduler var
          bEnSchedF6_ : BOOL := FALSE;
          wSchedWDHourStartF6_ : WORD; 
          wSchedWDMinStartF6_ : WORD; 
          wSchedWEHourStartF6_ : WORD; 
          wSchedWEMinStartF6_ : WORD;
          wSchedWDHourEndF6_ : WORD;
          wSchedWDMinEndF6_ : WORD;
          wSchedWEHourEndF6_ : WORD;
          wSchedWEMinEndF6_ : WORD;
          //unit var
          bUnitF6_ : ARRAY [1..22] OF BOOL;
      END_VAR


        // Reset trigger flag at minute change or at the exact scheduled time
        IF currM <> prevMinute OR 
           (currH = wSchedWDHourStartF6_ AND currM = wSchedWDMinStartF6_) OR 
           (currH = wSchedWDHourEndF6_ AND currM = wSchedWDMinEndF6_) THEN
            bUnitTriggered := FALSE;
            prevMinute := currM;
        END_IF

        // Unit Schedule Enable
        IF bEnSchedF6_ THEN
            // Weekday schedule
            IF currD >= 1 AND currD <= 5 THEN
                IF (wSchedWDHourStartF6_ <> wSchedWDHourEndF6_ OR wSchedWDMinStartF6_ <> wSchedWDMinEndF6_) THEN
                    // Schedule Unit ON
                    IF wSchedWDHourStartF6_ = currH AND wSchedWDMinStartF6_ = currM AND NOT bUnitTriggered THEN
                        bUnitTriggered := TRUE;
                        FOR i := 1 TO 22 DO
                            // Send command unit ON
                            IF bUnitF6_[i] THEN 
                                CASE i OF
                                    1: 
                                        
                                        FB_Bacnet.StartStopCommand_064.bEnWrite := TRUE;
                                        FB_Bacnet.StartStopCommand_064.bVal := TRUE;
                                    2: 
                                        
                                        FB_Bacnet.StartStopCommand_065.bEnWrite := TRUE;
                                        FB_Bacnet.StartStopCommand_065.bVal := TRUE;
                                    3: 
                                        
                                        FB_Bacnet.StartStopCommand_066.bEnWrite := TRUE;
                                        FB_Bacnet.StartStopCommand_066.bVal := TRUE;
                                    4: 
                                        
                                        FB_Bacnet.StartStopCommand_067.bEnWrite := TRUE;
                                        FB_Bacnet.StartStopCommand_067.bVal := TRUE;
                                    5: 
                                        
                                        FB_Bacnet.StartStopCommand_068.bEnWrite := TRUE;
                                        FB_Bacnet.StartStopCommand_068.bVal := TRUE;
                                    6: 
                                        
                                        FB_Bacnet.StartStopCommand_069.bEnWrite := TRUE;
                                        FB_Bacnet.StartStopCommand_069.bVal := TRUE;
                                    7: 
                                        
                                        FB_Bacnet.StartStopCommand_070.bEnWrite := TRUE;
                                        FB_Bacnet.StartStopCommand_070.bVal := TRUE;
                                    8: 
                                        
                                        FB_Bacnet.StartStopCommand_071.bEnWrite := TRUE;
                                        FB_Bacnet.StartStopCommand_071.bVal := TRUE;
                                    9: 
                                        
                                        FB_Bacnet.StartStopCommand_072.bEnWrite := TRUE;
                                        FB_Bacnet.StartStopCommand_072.bVal := TRUE;
                                    10: 
                                        
                                        FB_Bacnet.StartStopCommand_073.bEnWrite := TRUE;
                                        FB_Bacnet.StartStopCommand_073.bVal := TRUE;
                                    11: 
                                        
                                        FB_Bacnet.StartStopCommand_074.bEnWrite := TRUE;
                                        FB_Bacnet.StartStopCommand_074.bVal := TRUE;
                                    12: 
                                        
                                        FB_Bacnet.StartStopCommand_075.bEnWrite := TRUE;
                                        FB_Bacnet.StartStopCommand_075.bVal := TRUE;
                                    13: 
                                        
                                        FB_Bacnet.StartStopCommand_076.bEnWrite := TRUE;
                                        FB_Bacnet.StartStopCommand_076.bVal := TRUE;
                                    14: 
                                        
                                        FB_Bacnet.StartStopCommand_077.bEnWrite := TRUE;
                                        FB_Bacnet.StartStopCommand_077.bVal := TRUE;
                                    15: 
                                        
                                        FB_Bacnet.StartStopCommand_078.bEnWrite := TRUE;
                                        FB_Bacnet.StartStopCommand_078.bVal := TRUE;
                                    16: 
                                        
                                        FB_Bacnet.StartStopCommand_079.bEnWrite := TRUE;
                                        FB_Bacnet.StartStopCommand_079.bVal := TRUE;
                                    17: 
                                        
                                        FB_Bacnet.StartStopCommand_080.bEnWrite := TRUE;
                                        FB_Bacnet.StartStopCommand_080.bVal := TRUE;
                                    18: 
                                        
                                        FB_Bacnet.StartStopCommand_081.bEnWrite := TRUE;
                                        FB_Bacnet.StartStopCommand_081.bVal := TRUE;
                                    19: 
                                        
                                        FB_Bacnet.StartStopCommand_082.bEnWrite := TRUE;
                                        FB_Bacnet.StartStopCommand_082.bVal := TRUE;
                                    20: 
                                        
                                        FB_Bacnet.StartStopCommand_083.bEnWrite := TRUE;
                                        FB_Bacnet.StartStopCommand_083.bVal := TRUE;
                                    21: 
                                        
                                        FB_Bacnet.StartStopCommand_084.bEnWrite := TRUE;
                                        FB_Bacnet.StartStopCommand_084.bVal := TRUE;
                                    22: 
                                        
                                        FB_Bacnet_b.StartStopCommand_226.bEnWrite := TRUE;
                                        FB_Bacnet_b.StartStopCommand_226.bVal := TRUE;
                                END_CASE
                            END_IF
                        END_FOR
                    END_IF
                    // Schedule Unit OFF
                    IF wSchedWDHourEndF6_ = currH AND wSchedWDMinEndF6_ = currM AND NOT bUnitTriggered THEN
                        bUnitTriggered := TRUE;
                        FOR i := 1 TO 22 DO
                            // Send command unit OFF
                            IF bUnitF6_[i] THEN 
                                CASE i OF
                                    1: 
                                        
                                        FB_Bacnet.StartStopCommand_064.bEnWrite := TRUE;
                                        FB_Bacnet.StartStopCommand_064.bVal := FALSE;
                                    2: 
                                        
                                        FB_Bacnet.StartStopCommand_065.bEnWrite := TRUE;
                                        FB_Bacnet.StartStopCommand_065.bVal := FALSE;
                                    3: 
                                        
                                        FB_Bacnet.StartStopCommand_066.bEnWrite := TRUE;
                                        FB_Bacnet.StartStopCommand_066.bVal := FALSE;
                                    4: 
                                        
                                        FB_Bacnet.StartStopCommand_067.bEnWrite := TRUE;
                                        FB_Bacnet.StartStopCommand_067.bVal := FALSE;
                                    5: 
                                        
                                        FB_Bacnet.StartStopCommand_068.bEnWrite := TRUE;
                                        FB_Bacnet.StartStopCommand_068.bVal := FALSE;
                                    6: 
                                        
                                        FB_Bacnet.StartStopCommand_069.bEnWrite := TRUE;
                                        FB_Bacnet.StartStopCommand_069.bVal := FALSE;
                                    7: 
                                        
                                        FB_Bacnet.StartStopCommand_070.bEnWrite := TRUE;
                                        FB_Bacnet.StartStopCommand_070.bVal := FALSE;
                                    8: 
                                        
                                        FB_Bacnet.StartStopCommand_071.bEnWrite := TRUE;
                                        FB_Bacnet.StartStopCommand_071.bVal := FALSE;
                                    9: 
                                        
                                        FB_Bacnet.StartStopCommand_072.bEnWrite := TRUE;
                                        FB_Bacnet.StartStopCommand_072.bVal := FALSE;
                                    10: 
                                        
                                        FB_Bacnet.StartStopCommand_073.bEnWrite := TRUE;
                                        FB_Bacnet.StartStopCommand_073.bVal := FALSE;
                                    11: 
                                        
                                        FB_Bacnet.StartStopCommand_074.bEnWrite := TRUE;
                                        FB_Bacnet.StartStopCommand_074.bVal := FALSE;
                                    12: 
                                        
                                        FB_Bacnet.StartStopCommand_075.bEnWrite := TRUE;
                                        FB_Bacnet.StartStopCommand_075.bVal := FALSE;
                                    13: 
                                        
                                        FB_Bacnet.StartStopCommand_076.bEnWrite := TRUE;
                                        FB_Bacnet.StartStopCommand_076.bVal := FALSE;
                                    14: 
                                        
                                        FB_Bacnet.StartStopCommand_077.bEnWrite := TRUE;
                                        FB_Bacnet.StartStopCommand_077.bVal := FALSE;
                                    15: 
                                        
                                        FB_Bacnet.StartStopCommand_078.bEnWrite := TRUE;
                                        FB_Bacnet.StartStopCommand_078.bVal := FALSE;
                                    16: 
                                        
                                        FB_Bacnet.StartStopCommand_079.bEnWrite := TRUE;
                                        FB_Bacnet.StartStopCommand_079.bVal := FALSE;
                                    17: 
                                        
                                        FB_Bacnet.StartStopCommand_080.bEnWrite := TRUE;
                                        FB_Bacnet.StartStopCommand_080.bVal := FALSE;
                                    18: 
                                        
                                        FB_Bacnet.StartStopCommand_081.bEnWrite := TRUE;
                                        FB_Bacnet.StartStopCommand_081.bVal := FALSE;
                                    19: 
                                        
                                        FB_Bacnet.StartStopCommand_082.bEnWrite := TRUE;
                                        FB_Bacnet.StartStopCommand_082.bVal := FALSE;
                                    20: 
                                        
                                        FB_Bacnet.StartStopCommand_083.bEnWrite := TRUE;
                                        FB_Bacnet.StartStopCommand_083.bVal := FALSE;
                                    21: 
                                        
                                        FB_Bacnet.StartStopCommand_084.bEnWrite := TRUE;
                                        FB_Bacnet.StartStopCommand_084.bVal := FALSE;
                                    22: 
                                        
                                        FB_Bacnet_b.StartStopCommand_226.bEnWrite := TRUE;
                                        FB_Bacnet_b.StartStopCommand_226.bVal := FALSE;
                                END_CASE
                            END_IF
                        END_FOR
                    END_IF
                END_IF
            END_IF

            // Weekend schedule
            IF currD = 0 OR currD = 6 THEN
                IF (wSchedWEHourStartF6_ <> wSchedWEHourEndF6_ OR wSchedWEMinStartF6_ <> wSchedWEMinEndF6_) THEN
                    // Schedule Unit ON
                    IF wSchedWEHourStartF6_ = currH AND wSchedWEMinStartF6_ = currM AND NOT bUnitTriggered THEN
                        bUnitTriggered := TRUE;
                        FOR i := 1 TO 22 DO
                            // Send command unit ON
                            IF bUnitF6_[i] THEN 
                                CASE i OF
                                    1: 
                                        
                                        FB_Bacnet.StartStopCommand_064.bEnWrite := TRUE;
                                        FB_Bacnet.StartStopCommand_064.bVal := TRUE;
                                    2: 
                                        
                                        FB_Bacnet.StartStopCommand_065.bEnWrite := TRUE;
                                        FB_Bacnet.StartStopCommand_065.bVal := TRUE;
                                    3: 
                                        
                                        FB_Bacnet.StartStopCommand_066.bEnWrite := TRUE;
                                        FB_Bacnet.StartStopCommand_066.bVal := TRUE;
                                    4: 
                                        
                                        FB_Bacnet.StartStopCommand_067.bEnWrite := TRUE;
                                        FB_Bacnet.StartStopCommand_067.bVal := TRUE;
                                    5: 
                                        
                                        FB_Bacnet.StartStopCommand_068.bEnWrite := TRUE;
                                        FB_Bacnet.StartStopCommand_068.bVal := TRUE;
                                    6: 
                                        
                                        FB_Bacnet.StartStopCommand_069.bEnWrite := TRUE;
                                        FB_Bacnet.StartStopCommand_069.bVal := TRUE;
                                    7: 
                                        
                                        FB_Bacnet.StartStopCommand_070.bEnWrite := TRUE;
                                        FB_Bacnet.StartStopCommand_070.bVal := TRUE;
                                    8: 
                                        
                                        FB_Bacnet.StartStopCommand_071.bEnWrite := TRUE;
                                        FB_Bacnet.StartStopCommand_071.bVal := TRUE;
                                    9: 
                                        
                                        FB_Bacnet.StartStopCommand_072.bEnWrite := TRUE;
                                        FB_Bacnet.StartStopCommand_072.bVal := TRUE;
                                    10: 
                                        
                                        FB_Bacnet.StartStopCommand_073.bEnWrite := TRUE;
                                        FB_Bacnet.StartStopCommand_073.bVal := TRUE;
                                    11: 
                                        
                                        FB_Bacnet.StartStopCommand_074.bEnWrite := TRUE;
                                        FB_Bacnet.StartStopCommand_074.bVal := TRUE;
                                    12: 
                                        
                                        FB_Bacnet.StartStopCommand_075.bEnWrite := TRUE;
                                        FB_Bacnet.StartStopCommand_075.bVal := TRUE;
                                    13: 
                                        
                                        FB_Bacnet.StartStopCommand_076.bEnWrite := TRUE;
                                        FB_Bacnet.StartStopCommand_076.bVal := TRUE;
                                    14: 
                                        
                                        FB_Bacnet.StartStopCommand_077.bEnWrite := TRUE;
                                        FB_Bacnet.StartStopCommand_077.bVal := TRUE;
                                    15: 
                                        
                                        FB_Bacnet.StartStopCommand_078.bEnWrite := TRUE;
                                        FB_Bacnet.StartStopCommand_078.bVal := TRUE;
                                    16: 
                                        
                                        FB_Bacnet.StartStopCommand_079.bEnWrite := TRUE;
                                        FB_Bacnet.StartStopCommand_079.bVal := TRUE;
                                    17: 
                                        
                                        FB_Bacnet.StartStopCommand_080.bEnWrite := TRUE;
                                        FB_Bacnet.StartStopCommand_080.bVal := TRUE;
                                    18: 
                                        
                                        FB_Bacnet.StartStopCommand_081.bEnWrite := TRUE;
                                        FB_Bacnet.StartStopCommand_081.bVal := TRUE;
                                    19: 
                                        
                                        FB_Bacnet.StartStopCommand_082.bEnWrite := TRUE;
                                        FB_Bacnet.StartStopCommand_082.bVal := TRUE;
                                    20: 
                                        
                                        FB_Bacnet.StartStopCommand_083.bEnWrite := TRUE;
                                        FB_Bacnet.StartStopCommand_083.bVal := TRUE;
                                    21: 
                                        
                                        FB_Bacnet.StartStopCommand_084.bEnWrite := TRUE;
                                        FB_Bacnet.StartStopCommand_084.bVal := TRUE;
                                    22: 
                                        
                                        FB_Bacnet_b.StartStopCommand_226.bEnWrite := TRUE;
                                        FB_Bacnet_b.StartStopCommand_226.bVal := TRUE;
                                END_CASE
                            END_IF
                        END_FOR
                    END_IF
                    // Schedule Unit OFF
                    IF wSchedWEHourEndF6_ = currH AND wSchedWEMinEndF6_ = currM AND NOT bUnitTriggered THEN
                        bUnitTriggered := TRUE;
                        FOR i := 1 TO 22 DO
                            // Send command unit OFF
                            IF bUnitF6_[i] THEN 
                                CASE i OF
                                    1: 
                                        
                                        FB_Bacnet.StartStopCommand_064.bEnWrite := TRUE;
                                        FB_Bacnet.StartStopCommand_064.bVal := FALSE;
                                    2: 
                                        
                                        FB_Bacnet.StartStopCommand_065.bEnWrite := TRUE;
                                        FB_Bacnet.StartStopCommand_065.bVal := FALSE;
                                    3: 
                                        
                                        FB_Bacnet.StartStopCommand_066.bEnWrite := TRUE;
                                        FB_Bacnet.StartStopCommand_066.bVal := FALSE;
                                    4: 
                                        
                                        FB_Bacnet.StartStopCommand_067.bEnWrite := TRUE;
                                        FB_Bacnet.StartStopCommand_067.bVal := FALSE;
                                    5: 
                                        
                                        FB_Bacnet.StartStopCommand_068.bEnWrite := TRUE;
                                        FB_Bacnet.StartStopCommand_068.bVal := FALSE;
                                    6: 
                                        
                                        FB_Bacnet.StartStopCommand_069.bEnWrite := TRUE;
                                        FB_Bacnet.StartStopCommand_069.bVal := FALSE;
                                    7: 
                                        
                                        FB_Bacnet.StartStopCommand_070.bEnWrite := TRUE;
                                        FB_Bacnet.StartStopCommand_070.bVal := FALSE;
                                    8: 
                                        
                                        FB_Bacnet.StartStopCommand_071.bEnWrite := TRUE;
                                        FB_Bacnet.StartStopCommand_071.bVal := FALSE;
                                    9: 
                                        
                                        FB_Bacnet.StartStopCommand_072.bEnWrite := TRUE;
                                        FB_Bacnet.StartStopCommand_072.bVal := FALSE;
                                    10: 
                                        
                                        FB_Bacnet.StartStopCommand_073.bEnWrite := TRUE;
                                        FB_Bacnet.StartStopCommand_073.bVal := FALSE;
                                    11: 
                                        
                                        FB_Bacnet.StartStopCommand_074.bEnWrite := TRUE;
                                        FB_Bacnet.StartStopCommand_074.bVal := FALSE;
                                    12: 
                                        
                                        FB_Bacnet.StartStopCommand_075.bEnWrite := TRUE;
                                        FB_Bacnet.StartStopCommand_075.bVal := FALSE;
                                    13: 
                                        
                                        FB_Bacnet.StartStopCommand_076.bEnWrite := TRUE;
                                        FB_Bacnet.StartStopCommand_076.bVal := FALSE;
                                    14: 
                                        
                                        FB_Bacnet.StartStopCommand_077.bEnWrite := TRUE;
                                        FB_Bacnet.StartStopCommand_077.bVal := FALSE;
                                    15: 
                                        
                                        FB_Bacnet.StartStopCommand_078.bEnWrite := TRUE;
                                        FB_Bacnet.StartStopCommand_078.bVal := FALSE;
                                    16: 
                                        
                                        FB_Bacnet.StartStopCommand_079.bEnWrite := TRUE;
                                        FB_Bacnet.StartStopCommand_079.bVal := FALSE;
                                    17: 
                                        
                                        FB_Bacnet.StartStopCommand_080.bEnWrite := TRUE;
                                        FB_Bacnet.StartStopCommand_080.bVal := FALSE;
                                    18: 
                                        
                                        FB_Bacnet.StartStopCommand_081.bEnWrite := TRUE;
                                        FB_Bacnet.StartStopCommand_081.bVal := FALSE;
                                    19: 
                                        
                                        FB_Bacnet.StartStopCommand_082.bEnWrite := TRUE;
                                        FB_Bacnet.StartStopCommand_082.bVal := FALSE;
                                    20: 
                                        
                                        FB_Bacnet.StartStopCommand_083.bEnWrite := TRUE;
                                        FB_Bacnet.StartStopCommand_083.bVal := FALSE;
                                    21: 
                                        
                                        FB_Bacnet.StartStopCommand_084.bEnWrite := TRUE;
                                        FB_Bacnet.StartStopCommand_084.bVal := FALSE;
                                    22: 
                                        
                                        FB_Bacnet_b.StartStopCommand_226.bEnWrite := TRUE;
                                        FB_Bacnet_b.StartStopCommand_226.bVal := FALSE;
                                END_CASE
                            END_IF
                        END_FOR
                    END_IF
                END_IF
            END_IF
        END_IF

END_FUNCTION_BLOCK

// ---- POUs/FB_Scheduler/FB_Scheduler_F7.TcPOU

      FUNCTION_BLOCK FB_Scheduler_F7
      VAR_INPUT
          currH : WORD;
          currM : WORD;
          currD : WORD;
      END_VAR
      VAR_IN_OUT
          FB_Bacnet : FB_BACnet_DAIKIN_MasterStation_III_No_2;
          FB_Bacnet_b : FB_BACnet_DAIKIN_MasterStation_III_No_1;
      END_VAR
      VAR
          i : INT;
          bUnitTriggered : BOOL := FALSE; // New flag to track execution
          prevMinute : WORD := 0;        // New variable to track the previous minute
      END_VAR
      VAR PERSISTENT
          //scheduler var
          bEnSchedF7_ : BOOL := FALSE;
          wSchedWDHourStartF7_ : WORD; 
          wSchedWDMinStartF7_ : WORD; 
          wSchedWEHourStartF7_ : WORD; 
          wSchedWEMinStartF7_ : WORD;
          wSchedWDHourEndF7_ : WORD;
          wSchedWDMinEndF7_ : WORD;
          wSchedWEHourEndF7_ : WORD;
          wSchedWEMinEndF7_ : WORD;
          //unit var
          bUnitF7_ : ARRAY [1..24] OF BOOL;
      END_VAR


        // Reset trigger flag at minute change or at the exact scheduled time
        IF currM <> prevMinute OR 
           (currH = wSchedWDHourStartF7_ AND currM = wSchedWDMinStartF7_) OR 
           (currH = wSchedWDHourEndF7_ AND currM = wSchedWDMinEndF7_) THEN
            bUnitTriggered := FALSE;
            prevMinute := currM;
        END_IF

        // Unit Schedule Enable
        IF bEnSchedF7_ THEN
            // Weekday schedule
            IF currD >= 1 AND currD <= 5 THEN
                IF (wSchedWDHourStartF7_ <> wSchedWDHourEndF7_ OR wSchedWDMinStartF7_ <> wSchedWDMinEndF7_) THEN
                    // Schedule Unit ON
                    IF wSchedWDHourStartF7_ = currH AND wSchedWDMinStartF7_ = currM AND NOT bUnitTriggered THEN
                        bUnitTriggered := TRUE;
                        FOR i := 1 TO 24 DO
                            // Send command unit ON
                            IF bUnitF7_[i] THEN 
                                CASE i OF
                                    1: 
                                        
                                        FB_Bacnet.StartStopCommand_128.bEnWrite := TRUE;
                                        FB_Bacnet.StartStopCommand_128.bVal := TRUE;
                                    2: 
                                        
                                        FB_Bacnet.StartStopCommand_129.bEnWrite := TRUE;
                                        FB_Bacnet.StartStopCommand_129.bVal := TRUE;
                                    3: 
                                        
                                        FB_Bacnet.StartStopCommand_130.bEnWrite := TRUE;
                                        FB_Bacnet.StartStopCommand_130.bVal := TRUE;
                                    4: 
                                        
                                        FB_Bacnet.StartStopCommand_131.bEnWrite := TRUE;
                                        FB_Bacnet.StartStopCommand_131.bVal := TRUE;
                                    5: 
                                        
                                        FB_Bacnet.StartStopCommand_132.bEnWrite := TRUE;
                                        FB_Bacnet.StartStopCommand_132.bVal := TRUE;
                                    6: 
                                        
                                        FB_Bacnet.StartStopCommand_133.bEnWrite := TRUE;
                                        FB_Bacnet.StartStopCommand_133.bVal := TRUE;
                                    7: 
                                        
                                        FB_Bacnet.StartStopCommand_134.bEnWrite := TRUE;
                                        FB_Bacnet.StartStopCommand_134.bVal := TRUE;
                                    8: 
                                        
                                        FB_Bacnet.StartStopCommand_135.bEnWrite := TRUE;
                                        FB_Bacnet.StartStopCommand_135.bVal := TRUE;
                                    9: 
                                        
                                        FB_Bacnet.StartStopCommand_136.bEnWrite := TRUE;
                                        FB_Bacnet.StartStopCommand_136.bVal := TRUE;
                                    10: 
                                        
                                        FB_Bacnet.StartStopCommand_137.bEnWrite := TRUE;
                                        FB_Bacnet.StartStopCommand_137.bVal := TRUE;
                                    11: 
                                        
                                        FB_Bacnet.StartStopCommand_138.bEnWrite := TRUE;
                                        FB_Bacnet.StartStopCommand_138.bVal := TRUE;
                                    12: 
                                        
                                        FB_Bacnet.StartStopCommand_139.bEnWrite := TRUE;
                                        FB_Bacnet.StartStopCommand_139.bVal := TRUE;
                                    13: 
                                        
                                        FB_Bacnet.StartStopCommand_140.bEnWrite := TRUE;
                                        FB_Bacnet.StartStopCommand_140.bVal := TRUE;
                                    14: 
                                        
                                        FB_Bacnet.StartStopCommand_141.bEnWrite := TRUE;
                                        FB_Bacnet.StartStopCommand_141.bVal := TRUE;
                                    15: 
                                        
                                        FB_Bacnet.StartStopCommand_142.bEnWrite := TRUE;
                                        FB_Bacnet.StartStopCommand_142.bVal := TRUE;
                                    16: 
                                        
                                        FB_Bacnet.StartStopCommand_143.bEnWrite := TRUE;
                                        FB_Bacnet.StartStopCommand_143.bVal := TRUE;
                                    17: 
                                        
                                        FB_Bacnet.StartStopCommand_144.bEnWrite := TRUE;
                                        FB_Bacnet.StartStopCommand_144.bVal := TRUE;
                                    18: 
                                        
                                        FB_Bacnet.StartStopCommand_145.bEnWrite := TRUE;
                                        FB_Bacnet.StartStopCommand_145.bVal := TRUE;
                                    19: 
                                        
                                        FB_Bacnet.StartStopCommand_146.bEnWrite := TRUE;
                                        FB_Bacnet.StartStopCommand_146.bVal := TRUE;
                                    20: 
                                        
                                        FB_Bacnet.StartStopCommand_147.bEnWrite := TRUE;
                                        FB_Bacnet.StartStopCommand_147.bVal := TRUE;
                                    21: 
                                        
                                        FB_Bacnet.StartStopCommand_148.bEnWrite := TRUE;
                                        FB_Bacnet.StartStopCommand_148.bVal := TRUE;
                                    22: 
                                        
                                        FB_Bacnet.StartStopCommand_176.bEnWrite := TRUE;
                                        FB_Bacnet.StartStopCommand_176.bVal := TRUE;
                                    23: 
                                        
                                        FB_Bacnet_b.StartStopCommand_241.bEnWrite := TRUE;
                                        FB_Bacnet_b.StartStopCommand_241.bVal := TRUE;
                                    24: 
                                        
                                        FB_Bacnet_b.StartStopCommand_227.bEnWrite := TRUE;
                                        FB_Bacnet_b.StartStopCommand_227.bVal := TRUE;
                                END_CASE
                            END_IF
                        END_FOR
                    END_IF
                    // Schedule Unit OFF
                    IF wSchedWDHourEndF7_ = currH AND wSchedWDMinEndF7_ = currM AND NOT bUnitTriggered THEN
                        bUnitTriggered := TRUE;
                        FOR i := 1 TO 24 DO
                            // Send command unit OFF
                            IF bUnitF7_[i] THEN 
                                CASE i OF
                                    1: 
                                        
                                        FB_Bacnet.StartStopCommand_128.bEnWrite := TRUE;
                                        FB_Bacnet.StartStopCommand_128.bVal := FALSE;
                                    2: 
                                        
                                        FB_Bacnet.StartStopCommand_129.bEnWrite := TRUE;
                                        FB_Bacnet.StartStopCommand_129.bVal := FALSE;
                                    3: 
                                        
                                        FB_Bacnet.StartStopCommand_130.bEnWrite := TRUE;
                                        FB_Bacnet.StartStopCommand_130.bVal := FALSE;
                                    4: 
                                        
                                        FB_Bacnet.StartStopCommand_131.bEnWrite := TRUE;
                                        FB_Bacnet.StartStopCommand_131.bVal := FALSE;
                                    5: 
                                        
                                        FB_Bacnet.StartStopCommand_132.bEnWrite := TRUE;
                                        FB_Bacnet.StartStopCommand_132.bVal := FALSE;
                                    6: 
                                        
                                        FB_Bacnet.StartStopCommand_133.bEnWrite := TRUE;
                                        FB_Bacnet.StartStopCommand_133.bVal := FALSE;
                                    7: 
                                        
                                        FB_Bacnet.StartStopCommand_134.bEnWrite := TRUE;
                                        FB_Bacnet.StartStopCommand_134.bVal := FALSE;
                                    8: 
                                        
                                        FB_Bacnet.StartStopCommand_135.bEnWrite := TRUE;
                                        FB_Bacnet.StartStopCommand_135.bVal := FALSE;
                                    9: 
                                        
                                        FB_Bacnet.StartStopCommand_136.bEnWrite := TRUE;
                                        FB_Bacnet.StartStopCommand_136.bVal := FALSE;
                                    10: 
                                        
                                        FB_Bacnet.StartStopCommand_137.bEnWrite := TRUE;
                                        FB_Bacnet.StartStopCommand_137.bVal := FALSE;
                                    11: 
                                        
                                        FB_Bacnet.StartStopCommand_138.bEnWrite := TRUE;
                                        FB_Bacnet.StartStopCommand_138.bVal := FALSE;
                                    12: 
                                        
                                        FB_Bacnet.StartStopCommand_139.bEnWrite := TRUE;
                                        FB_Bacnet.StartStopCommand_139.bVal := FALSE;
                                    13: 
                                        
                                        FB_Bacnet.StartStopCommand_140.bEnWrite := TRUE;
                                        FB_Bacnet.StartStopCommand_140.bVal := FALSE;
                                    14: 
                                        
                                        FB_Bacnet.StartStopCommand_141.bEnWrite := TRUE;
                                        FB_Bacnet.StartStopCommand_141.bVal := FALSE;
                                    15: 
                                        
